// TIA Portal V19 export
TYPE "LEXCHANGETRAY_typeConstraintRollerEm_toHandlingXyzRecieve"
// stored: Access Published
   STRUCT
      feedback { S7_SetPoint := 'True'} : "LEXCHANGETRAY_typeHandlingXyzEm_toConstraintRollerFeedback";
      req { S7_SetPoint := 'True'} : "LEXCHANGETRAY_typeHandlingXyzEm_toConstraintRollerReq";
   END_STRUCT;
END_TYPE
